// TIA Portal V19 export
VAR_GLOBAL   // PLC tag table "IPC_MSG_KEYS_CONST"
END_VAR
VAR_GLOBAL CONSTANT   // user constants
   LOG_KEY_SEPARATOR : String := ';';
   LOG_PAR_CHANGE_KEY_PAR_NUM : String := '[numero parametro]=';
   LOG_PAR_CHANGE_KEY_PAR_DESC : String := '[descrizione parametro]=';
   LOG_PAR_CHANGE_KEY_UM : String := '[unita di misura]=';
   LOG_PAR_CHANGE_KEY_VALUE_PRV : String := '[valore precedente]=';
   LOG_PAR_CHANGE_KEY_VALUE_ACT : String := '[valore attuale]=';
   LOG_PAR_CHANGE_KEY_PAR_GROUP : String := '[Gruppo parametri]=';
END_VAR
